// TwinCAT 3 PLC project plc1
// ProgramVersion: 3.1.4023.0
// libraries:
//   Tc2_Standard, * (Beckhoff Automation GmbH)
//   Tc2_System, * (Beckhoff Automation GmbH)
//   Tc2_Utilities, * (Beckhoff Automation GmbH)
//   Tc3_Module, * (Beckhoff Automation GmbH)
//   VisuDialogs, * (System)
// project tree:
//   DUTs/ ST_Event.TcDUT
//   / FasterTask.TcTTO, GlobalTextList.TcGTLO, PlcTask.TcTTO, Visualization Manager.TcVMO (not stored)
//   GVLs/ GVL.TcGVL
//   POUs/FBs/ FB_Cylinder.TcPOU, FB_ScaleAnalogInput.TcPOU, FB_ScaleAnalogoutput.TcPOU
//   POUs/CylPrograms/ Module1Control.TcPOU
//   POUs/ MAIN.TcPOU
//   VISUs/ Visualization.TcVIS
// real-time tasks:
//   TASK FasterTask: cycle T#1ms, priority 1, ADS port 350
//   TASK PlcTask: cycle T#5ms, priority 20, ADS port 351

CONFIGURATION plc1
    RESOURCE PLC ON TwinCAT3
        TASK FasterTask(INTERVAL := T#1ms, PRIORITY := 1);
        TASK PlcTask(INTERVAL := T#5ms, PRIORITY := 20);
        PROGRAM Module1Control WITH FasterTask : Module1Control;
        PROGRAM MAIN WITH PlcTask : MAIN;
    END_RESOURCE
END_CONFIGURATION

// ---- DUTs/ST_Event.TcDUT
TYPE ST_Event :
STRUCT
	sDateTime		: STRING;
	sEvent			: STRING;
	fProcVal		: REAL;
	bHeaterState	: BOOL;
END_STRUCT
END_TYPE

// ---- GVLs/GVL.TcGVL
{attribute 'qualified_only'}
VAR_GLOBAL
END_VAR

// ---- POUs/CylPrograms/Module1Control.TcPOU
PROGRAM Module1Control
VAR
	//Cyl1
	FB_Cylinder_Right: FB_Cylinder;
	ExtendCyl_Right: BOOL;
	Cyl_RightStatus: BOOL;
	
	//Poti 
	Poti_Scale: FB_ScaleAnalogInput;
	Poti_in AT %I* : DINT;
	{attribute 'OPC.UA.DA' := '1'}
	{attribute 'TcAnalytics'}
	Display AT %Q*:INT;
	
	
	
	FB_Cylinder_Left: FB_Cylinder;
	ExtendCyl_Left: BOOL;
	Cyl_LeftStatus: BOOL;
END_VAR

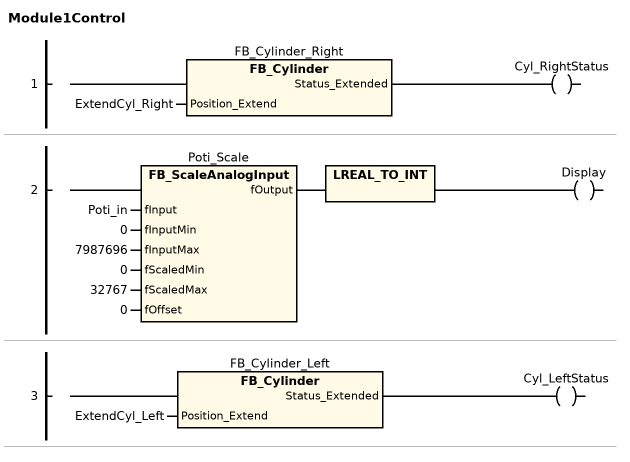
// NETWORK 1
FB_Cylinder_Right(Position_Extend := ExtendCyl_Right); // FB_Cylinder
Cyl_RightStatus := FB_Cylinder_Right.Status_Extended;

// NETWORK 2
Poti_Scale(
    fInput := Poti_in,
    fInputMin := 0,
    fInputMax := 7987696,
    fScaledMin := 0,
    fScaledMax := 32767,
    fOffset := 0); // FB_ScaleAnalogInput
Display := LREAL_TO_INT(Poti_Scale.fOutput);

// NETWORK 3
FB_Cylinder_Left(Position_Extend := ExtendCyl_Left); // FB_Cylinder
Cyl_LeftStatus := FB_Cylinder_Left.Status_Extended;

END_PROGRAM

// ---- POUs/FBs/FB_Cylinder.TcPOU
FUNCTION_BLOCK FB_Cylinder
VAR_INPUT
	Position_Extend: BOOL;
END_VAR
VAR_OUTPUT
	Status_Extended:BOOL;
END_VAR
VAR
	CylinderOutput AT %Q*:BOOL;
END_VAR

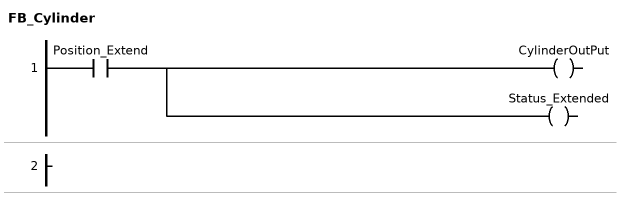
// NETWORK 1
CylinderOutPut := Position_Extend;
Status_Extended := Position_Extend;

// NETWORK 2

END_FUNCTION_BLOCK

// ---- POUs/FBs/FB_ScaleAnalogInput.TcPOU
FUNCTION_BLOCK FB_ScaleAnalogInput
VAR_INPUT
	///Actual value
	fInput: LREAL;
	///Min 'actual value' can be
	fInputMin: LREAL;
	///Max 'actual value' can be (analog will be 32768)
	fInputMax: LREAL;
	///Scaled Units MIN
	fScaledMin: LREAL;
	///Scaled Units MAX
	fScaledMax: LREAL;
	///Offset shift (if any)
	fOffset: LREAL;
END_VAR
VAR_OUTPUT
	///Actual value in 'Engineering Units'
	fOutput: LREAL;
END_VAR

fOutput := (fInput - fInputMin)*(fScaledMax - fScaledMin)/(fInputMax - fInputMin) + fScaledMin + fOffset;

END_FUNCTION_BLOCK

// ---- POUs/MAIN.TcPOU
PROGRAM MAIN
VAR
	stEventArray	: ARRAY[0..iNumEvents] OF ST_Event;
	
	
	bEstop			: BOOL :=TRUE;
	{attribute 'OPC.UA.DA' := '1'}
	bRun			: BOOL;
	{attribute 'TcAnalytics'}
	{attribute 'OPC.UA.DA' := '1'}
	rRealVal		: REAL;  //Process Value
	{attribute 'TcAnalytics'}
	bHeater			: BOOL;
	
	fbTON			: TON;
	{attribute 'TcAnalytics'}
	{attribute 'OPC.UA.DA' := '1'}
	bGoodCpk		: BOOL :=TRUE;
	lrRandom		: LREAL;
	iTmrPreset		: INT :=1000;
	iTmrET			: INT;
	fbDRAND			: DRAND;	
	rDutyCycle		: REAL :=50;

	sState			: STRING;
	sPrevState		: STRING;
	
	// date/time vars
    fbGetSystemTime  	: GETSYSTEMTIME;
    fileTimeUTC         : T_FILETIME;
    sDateTimeUTC        : STRING[32];

    fileTimeLocal       : T_FILETIME;
	systemTimeLocal		: TIMESTRUCT;
	sDateTimeLocal		: STRING[32];
	
	ulSysTime			: ULINT;

	myTime: DATE_AND_TIME;
	myTime2: TIME;
	myTime3: LTIME;
END_VAR

VAR CONSTANT
	iNumEvents: UINT := 99;
END_VAR

IF bEstop THEN
	bRun := FALSE;
	rRealVal := 50.0;
	bHeater := FALSE;
ELSE
	// run virtual machine
	IF bRun THEN
		fbDRAND(Seed:= iTmrET, Num=> lrRandom);
				
		IF bGoodCpk THEN
			rRealVal := 50 + 10 *(LREAL_TO_REAL(lrRandom)-0.5);
		ELSE
			rRealVal := rRealVal + 2 *(LREAL_TO_REAL(lrRandom)-0.5);
		END_IF
	END_IF	

	// Cycle heater based on duty cycle 	
	fbTON(IN:=NOT fbTON.q , PT:=INT_TO_TIME(iTmrPreset) , Q=> , ET=> );	
	iTmrET := TIME_TO_INT(fbTON.ET);
	
	IF iTmrET < iTmrPreset*rDutyCycle/100 THEN
		bHeater := TRUE;
	ELSE
		bHeater := FALSE;
	END_IF


END_IF

// Call EventLog action
aEventLog();

ACTION aEventLog:
// get timestamp
fbGetSystemTime(timeLoDW=>fileTimeUTC.dwLowDateTime, timeHiDW=>fileTimeUTC.dwHighDateTime);	// returns UTC time
sDateTimeUTC := SYSTEMTIME_TO_STRING(FILETIME_TO_SYSTEMTIME(fileTimeUTC));

// adjust for local timezone
//fileTimeLocal := F_TranslateFileTimeBias(in:= fileTime, bias:= WEST_EUROPE_TZI.bias + WEST_EUROPE_TZI.daylightBias, toUTC:= FALSE);
fileTimeLocal := F_TranslateFileTimeBias(in:= fileTimeUTC, bias:= 6*60, toUTC:= FALSE);
systemTimeLocal:=FILETIME_TO_SYSTEMTIME(fileTimeLocal);
sDateTimeLocal := SYSTEMTIME_TO_STRING(systemTimeLocal);

ulSysTime:=F_GetSystemTime();	// how to convert to string??

//Daymon playtime...
myTime := ULINT_TO_DT(ulSysTime);
myTime2 := ULINT_TO_TIME(ulSysTime);
myTime3 := ULINT_TO_LTIME(ulSysTime);


IF bEstop THEN
	sState := 'E-Stopped';
ELSE
	sState := 'Idle';	// default state if no Estop
	IF bRun THEN
		sState := 'Running';

		// ALARM - process out of spec - stop
		IF (rRealVal < 10) OR (rRealVal > 90) THEN
			bRun := FALSE;
			sState := 'Stopped - Out of Spec - Low!';
		END_IF
		IF (rRealVal > 90) THEN
			bRun := FALSE;
			sState := 'Stopped - Out of Spec - Hi!';
		END_IF

		// WARNING - process Cpk bad - but continue running
		IF sState = 'Running' THEN
			IF (rRealVal < 30) THEN
				sState := 'Running Low - Check Process!';
			END_IF
			IF (rRealVal > 70) THEN
				sState := 'Running High - Check Process!';
			END_IF
		END_IF
	END_IF
END_IF

(* Manage Event array... *)
IF sState <> sPrevState THEN	// if state change shift data down and add new event to top
	MEMMOVE(destAddr:= ADR(stEventArray[1]), srcAddr:= ADR(stEventArray[0]), n:= SIZEOF(stEventArray[0])*iNumEvents);

	(* current event values *)
	stEventArray[0].sDateTime := sDateTimeLocal;
	stEventArray[0].sEvent := sState;
	stEventArray[0].fProcVal := rRealVal;
	stEventArray[0].bHeaterState := bHeater;
END_IF
sPrevState := sState;
END_ACTION

END_PROGRAM

// ---- POUs/FBs/FB_ScaleAnalogoutput.TcPOU
FUNCTION_BLOCK FB_ScaleAnalogoutput
VAR_INPUT
	///Engineering Units Input
	fInput: LREAL;
	///Min 'Engineering Units' can be
	fInputMin: LREAL;
	///Max 'Engineering Units' can be (analog will be 32768)
	fInputMax: LREAL;
	///Analog value MIN (DEC 16 bit)
	fOutputMin: INT;
	///Analog value MAX (DEC 16 bit)
	fOutputMax: INT;
END_VAR
VAR_OUTPUT
	///Scaled value to be sent to Analog module (EL4xxx)
	nOutput: INT;
END_VAR
VAR
	///Internal var
	fTemp: LREAL;
END_VAR

IF fInput >fInputMax THEN
	nOutput := fOutputMax;
ELSIF fInput < fOutputMin THEN
	nOutput := fOutputMin;
ELSE
	nOutput := LREAL_TO_INT( (fInput - fInputMin)*(fOutputMax - fOutputMin)/(fInputMax - fInputMin) + fOutputMin);
END_IF

END_FUNCTION_BLOCK

// ---- GlobalTextList.TcGTLO
TEXTLIST GlobalTextList
  285 = '%0.3f'
  240 = '%s'
  53 = '(click to chg)'
  289 = '(Setpoint = 50)'
  288 = 'Bad Cpk'
  807 = 'DateTime'
  239 = 'Estop'
  948 = 'Event'
  287 = 'Good Cpk'
  54 = 'Heater'
  425 = 'Heater Duty Cycle % = %1.2f'
  371 = 'Heater State'
  825 = 'Process Value'
  286 = 'Process var'
  284 = 'Run / Stop'
  52 = 'Timer Preset'
END_TEXTLIST

// ---- VISUs/Visualization.TcVIS
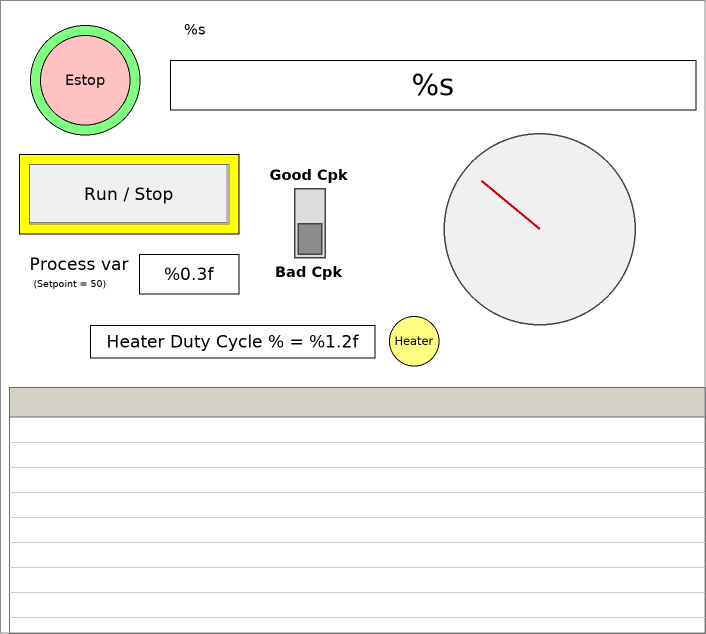
VISUALIZATION Visualization  // 706x634
    Rectangle (265,158 87x34), "Good Cpk"
    Ellipse (30,25 110x110), colour toggle: MAIN.bEstop
    Ellipse (40,35 90x90), "Estop"
        toggle MAIN.bEstop
    Rectangle (170,60 526x50), "%s", text variable: MAIN.sState
    Rectangle (181,17 255x25), "%s", text variable: MAIN.sDateTimeLocal
    Rectangle (19,154 220x80), colour toggle: MAIN.bRun
    Button (29,164 200x60), "Run / Stop", pressed state: MAIN.bRun
        toggle MAIN.bRun
    Rectangle (139,254 100x40), "%0.3f", text variable: MAIN.rRealVal
        OnMouseDown: write the text variable via VisuDialogs.Keypad
    Rectangle (14,249 130x30), "Process var"
    Rectangle (34,269 75x30), "(Setpoint = 50)"
    Meter180 (375,133 329x192), value: MAIN.rRealVal, style: Meter-Meter180-Gray, scale format: %.1f, scale 0..100
    Rectangle (90,325 285x33), "Heater Duty Cycle % = %1.2f", text variable: MAIN.rDutyCycle
        OnMouseDown: write the text variable via VisuDialogs.Numpad, min 1, max 100
    Ellipse (389,316 50x50), "Heater", colour toggle: MAIN.bHeater
    Table (9,387 697x247), data array: MAIN.stEventArray
        p3854506369: MAIN.stEventArray[INDEX].sDateTime
        p1892666644: MAIN.stEventArray[INDEX].sEvent
        p338671338: MAIN.stEventArray[INDEX].fProcVal
        p1755163831: Process Value
        p1128707560: MAIN.iNumEvents
        p2170511999: MAIN.stEventArray[INDEX].bHeaterState
        p4092479075: Heater State
    Rectangle (265,255 87x34), "Bad Cpk"
    DipSwitch (275,188 70x70), variable: MAIN.bGoodCpk, behaviour: TOGGLE, style: Switch-DipSwitch-Gray
END_VISUALIZATION
